{attribute 'linkalways'} 
{attribute 'no_explicit_call' := 'This FB is a CLASS and must be accessed using methods or properties'}
{attribute 'enable_dynamic_creation'}
FUNCTION_BLOCK _ETcVnBlobCombination EXTENDS EnumDatatypeBase
VAR
	localData : ETcVnBlobCombination;
	activeData : REFERENCE TO ETcVnBlobCombination;
	enumBaseDatatype : _DINT(localData);
END_VAR

METHOD PRIVATE AddLocalEnumeration
VAR_INPUT
	Enumeration : T_MAXSTRING;
	Value : ETcVnBlobCombination;
END_VAR
AddEnumeration(Enumeration, Value);
END_METHOD

PROPERTY PUBLIC Address : PVOID
GET
Address := ADR(activeData);
END_GET
END_PROPERTY

METHOD PUBLIC ClearReference
VAR_INPUT
END_VAR
activeData REF= localData;
SetBaseDatatypeReference();
END_METHOD

METHOD PUBLIC Clone : I_Datatype
VAR
    pClone : POINTER TO _ETcVnBlobCombination;
END_VAR
pClone := __NEW(_ETcVnBlobCombination(InitialValue := Value));
Clone := pClone^;
END_METHOD

METHOD FB_init : BOOL
VAR_INPUT
	bInitRetains : BOOL; // if TRUE, the retain variables are initialized (warm start / cold start)
	bInCopyCode : BOOL;  // if TRUE, the instance afterwards gets moved into the copy code (online change)
	InitialValue : ETcVnBlobCombination;
END_VAR
localData := InitialValue;
AddBaseDatatype(enumBaseDatatype);
ClearReference();

AddLocalEnumeration('TCVN_BC_SMALLEST', ETcVnBlobCombination.TCVN_BC_SMALLEST);
AddLocalEnumeration('TCVN_BC_LARGEST', ETcVnBlobCombination.TCVN_BC_LARGEST);
AddLocalEnumeration('TCVN_BC_MIN_THRESHOLD', ETcVnBlobCombination.TCVN_BC_MIN_THRESHOLD);
AddLocalEnumeration('TCVN_BC_MAX_THRESHOLD', ETcVnBlobCombination.TCVN_BC_MAX_THRESHOLD);
AddLocalEnumeration('TCVN_BC_MEDIAN_THRESHOLD', ETcVnBlobCombination.TCVN_BC_MEDIAN_THRESHOLD);
END_METHOD

PROPERTY PUBLIC Identifier : T_MAXSTRING
GET
Identifier := 'ETcVnBlobCombination';
END_GET
END_PROPERTY

METHOD IsEnumeratorValueEqual : BOOL
VAR_INPUT
	Enumerator : I_KeyValueForwardEnumerator;
END_VAR
VAR
	storedValue : ETcVnBlobCombination;
END_VAR
IF NOT Enumerator.TryGet(storedValue) THEN
	RETURN;
END_IF

IsEnumeratorValueEqual := storedValue = activeData;
END_METHOD

METHOD PUBLIC MakeReferenceTo
VAR_INPUT
	ReferenceTarget : REFERENCE TO ETcVnBlobCombination;
END_VAR
activeData REF= ReferenceTarget;
SetBaseDatatypeReference();
END_METHOD

METHOD PROTECTED SetBaseDatatypeReference
VAR_INPUT
END_VAR
enumBaseDatatype.MakeReferenceTo(activeData);
END_METHOD

PROPERTY PUBLIC Size : UDINT
GET
Size := SIZEOF(activeData);
END_GET
END_PROPERTY

METHOD TryMakeReferenceTo : BOOL
VAR_INPUT
	Target : I_Datatype;
END_VAR
VAR
	targetAsEnum : I_EnumDatatype;
	pTargetData : POINTER TO ETcVnBlobCombination;
END_VAR
IF NOT Target.TryResolveAsEnumDatatype(targetAsEnum) THEN
	RETURN;
END_IF

IF targetAsEnum.Identifier <> Identifier THEN
	RETURN;
END_IF

pTargetData := Target.Address;
activeData REF= pTargetData^;
SetBaseDatatypeReference();
TryMakeReferenceTo := TRUE;
END_METHOD

PROPERTY PUBLIC Value : ETcVnBlobCombination
GET
Value := activeData;
END_GET
SET
activeData := Value;
END_SET
END_PROPERTY

END_FUNCTION_BLOCK

(* stored: Version 1.1.0.1, ProductVersion 3.1.4024.12
   POU _ETcVnBlobCombination: Id {ca317810-447f-079b-288b-88f3f5bf9858}, SpecialFunc None
   Folder Constructor: Id {1882b504-220f-0b49-13d1-0720b479204a}
   Folder Private: Id {e48e4a31-db4a-0fa1-0303-d2dac75f2a17}
   Folder Protected: Id {4aac66e6-3e55-01e7-17ea-be29b9d478a3}
   Method AddLocalEnumeration: Id {d376e38b-ad98-003e-12db-7a88ba7f75d1}
   Property Address: Id {18e32ca1-1536-0c89-2b98-81648bd01222}
   Get Get: Id {cb245e6b-c7c9-0c42-1432-5aec5e1b7a46}
   Method ClearReference: Id {5126681f-fe8f-0dba-3de8-2e0f4b18e786}
   Method Clone: Id {34cd77a5-3ca4-0c75-3e59-70c98477eed6}
   Method FB_init: Id {837f7f22-3b0b-000f-1261-49711579d085}
   Property Identifier: Id {c084283e-0ce0-0367-3ae8-fa79a52ab26e}
   Get Get: Id {110a443a-2753-0b63-22f6-c9ebaaaf3e14}
   Method IsEnumeratorValueEqual: Id {82f70e1a-e023-0b2b-3374-e1aee8e451cb}
   Method MakeReferenceTo: Id {41b41418-f854-0079-2bc2-09c149c6161d}
   Method SetBaseDatatypeReference: Id {9acb2d84-59f2-008b-070d-41ed1ed344cf}
   Property Size: Id {749d2786-edc3-0423-30ee-535ae22601c9}
   Get Get: Id {468fe52f-a72d-038a-3e5e-1dc32b8ece78}
   Method TryMakeReferenceTo: Id {0639b0e2-e02d-0216-0c27-e9350e0f41e3}
   Property Value: Id {c93b5027-134f-0bd2-1438-961fcb94b3e4}
   Get Get: Id {61302c6c-2b66-00b3-06af-26c176fd53b0}
   Set Set: Id {4cd8847e-d019-09f2-0535-6dfcb341eff6} *)
